Staubli VAL3: setMenu.pgx

public program setMenu(string& x_sMenuName[], bool x_bShowName, num x_nY)
// Show the
  local num i
begin
  //
  // usage
  // menuname"choice1,choise2,..choise7,choice8"
  //
  // the page will start from the y- line
  //
  //
  if size(x_sMenuName)<10
    for i=0 to (size(x_sMenuName)-1)
      if x_sMenuName[i]!="" and x_sMenuName[i]!=" "
        if x_bShowName==false
          call typeMenu(i+1,"F"+toString("1",i+1))
        else
          call typeMenu(i+1,x_sMenuName[i])
        endIf
        if x_nY!=-1
          call type(0,i+x_nY,("F"+(toString("1",i+1)+" "+x_sMenuName[i])))
        endIf
      endIf
    endFor
  endIf
end
